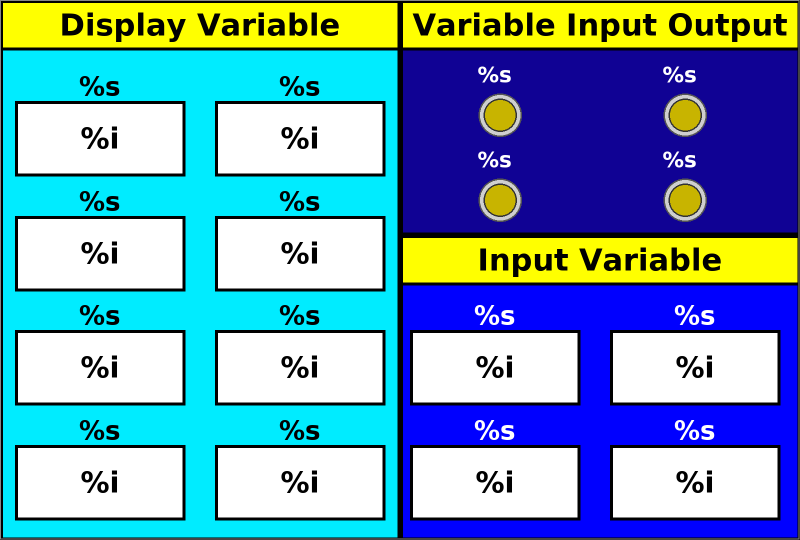
VISUALIZATION Screen_Rinse  // 800x540
    Rectangle (400,0 400x235)
    Rectangle (400,235 400x305)
    Rectangle (0,0 400x540)
    Rectangle (15,69 170x35), "%s", text variable: GVL.HMI_Rinse_Name_Display[0]
    Rectangle (15,101 170x75), "%i", text variable: GVL.HMI_Rinse_Display_Var[0]
    Rectangle (215,69 170x35), "%s", text variable: GVL.HMI_Rinse_Name_Display[1]
    Rectangle (215,101 170x75), "%i", text variable: GVL.HMI_Rinse_Display_Var[1]
    Rectangle (15,184 170x35), "%s", text variable: GVL.HMI_Rinse_Name_Display[2]
    Rectangle (15,216 170x75), "%i", text variable: GVL.HMI_Rinse_Display_Var[2]
    Rectangle (215,184 170x35), "%s", text variable: GVL.HMI_Rinse_Name_Display[3]
    Rectangle (215,216 170x75), "%i", text variable: GVL.HMI_Rinse_Display_Var[3]
    Rectangle (15,298 170x35), "%s", text variable: GVL.HMI_Rinse_Name_Display[4]
    Rectangle (15,330 170x75), "%i", text variable: GVL.HMI_Rinse_Display_Var[4]
    Rectangle (215,298 170x35), "%s", text variable: GVL.HMI_Rinse_Name_Display[5]
    Rectangle (215,330 170x75), "%i", text variable: GVL.HMI_Rinse_Display_Var[5]
    Rectangle (15,413 170x35), "%s", text variable: GVL.HMI_Rinse_Name_Display[6]
    Rectangle (15,445 170x75), "%i", text variable: GVL.HMI_Rinse_Display_Var[6]
    Rectangle (215,413 170x35), "%s", text variable: GVL.HMI_Rinse_Name_Display[7]
    Rectangle (215,445 170x75), "%i", text variable: GVL.HMI_Rinse_Display_Var[7]
    Rectangle (410,298 170x35), "%s", text variable: GVL.HMI_Rinse_Name_Input[0]
    Rectangle (410,330 170x75), "%i", text variable: GVL.HMI_Rinse_Input_Var[0]
        OnMouseClick: write GVL.HMI_Rinse_Input_Var[0] via VisuDialogs.Numpad
    Rectangle (610,298 170x35), "%s", text variable: GVL.HMI_Rinse_Name_Input[1]
    Rectangle (610,330 170x75), "%i", text variable: GVL.HMI_Rinse_Input_Var[1]
        OnMouseClick: write GVL.HMI_Rinse_Input_Var[1] via VisuDialogs.Numpad
    Rectangle (410,413 170x35), "%s", text variable: GVL.HMI_Rinse_Name_Input[2]
    Rectangle (410,445 170x75), "%i", text variable: GVL.HMI_Rinse_Input_Var[2]
        OnMouseClick: write GVL.HMI_Rinse_Input_Var[2] via VisuDialogs.Numpad
    Rectangle (610,413 170x35), "%s", text variable: GVL.HMI_Rinse_Name_Input[3]
    Rectangle (610,445 170x75), "%i", text variable: GVL.HMI_Rinse_Input_Var[3]
        OnMouseClick: write GVL.HMI_Rinse_Input_Var[3] via VisuDialogs.Numpad
    Rectangle (410,60 170x30), "%s", text variable: GVL.HMI_Rinse_Name_IO[0]
    Rectangle (595,60 170x30), "%s", text variable: GVL.HMI_Rinse_Name_IO[1]
    Rectangle (410,145 170x30), "%s", text variable: GVL.HMI_Rinse_Name_IO[2]
    Rectangle (595,145 170x30), "%s", text variable: GVL.HMI_Rinse_Name_IO[3]
    Rectangle (0,0 400x50), "Display Variable"
    Rectangle (400,0 400x50), "Variable Input Output"
    Rectangle (400,235 400x50), "Input Variable"
    Lamp1 (475,90 50x50), variable: GVL.HMI_Rinse_IO_Var[0], style: Lamp-Lamp1-Yellow
    Lamp1 (660,90 50x50), variable: GVL.HMI_Rinse_IO_Var[1], style: Lamp-Lamp1-Yellow
    Lamp1 (660,175 50x50), variable: GVL.HMI_Rinse_IO_Var[3], style: Lamp-Lamp1-Yellow
    Lamp1 (475,175 50x50), variable: GVL.HMI_Rinse_IO_Var[2], style: Lamp-Lamp1-Yellow
END_VISUALIZATION

(* stored: Version 1.1.0.1, ProductVersion 3.1.4024.12
   Visu Screen_Rinse: Id {aae57c7c-e003-4921-8de3-70791a134445} *)
